(* PLC project tipper, Dassault Systèmes ControlBuild 2024x *)
(* stored: creationDateTime 2023-10-03T11:12:52-01:00 *)

(* This module simulates the behaviour of a tipper. It takes a rotation speed as input and can move actors and products that are in interaction. *)
FUNCTION_BLOCK equipment_library.tipper
  VAR_INPUT
    rotationSpeed : REAL := 0.0;
  END_VAR
  VAR_OUTPUT
    angleRotationRad : REAL := 0.0;
    incRotation : REAL := 0.0;
    angleRotationDeg : REAL := 0.0;
  END_VAR
  VAR
    status_act_prod : DINT := 0;
    m11 : REAL := 1.0;
    m12 : REAL := 0.0;
    m13 : REAL := 0.0;
    m14 : REAL := 0.0;
    m21 : REAL := 0.0;
    m22 : REAL := 1.0;
    m23 : REAL := 0.0;
    m24 : REAL := 0.0;
    m31 : REAL := 0.0;
    m32 : REAL := 0.0;
    m33 : REAL := 1.0;
    m34 : REAL := 0.0;
    m41 : REAL := 0.0;
    m42 : REAL := 0.0;
    m43 : REAL := 0.0;
    m44 : REAL := 1.0;
    incrementRotation : REAL := 0.0;
    initPosX : REAL := 0.0;
    initPosY : REAL := 0.0;
    initPosZ : REAL := 0.0;
    firstCycle : BOOL := false;
  END_VAR
  VAR CONSTANT
    fixedPositions : ARRAY[1..5] OF REAL := [0.0, 90.0, 180.0, 270.0, 360.0];
    deltaPos : REAL(0.0..45.0) := 15.0;
  END_VAR
  VAR
    d_locking : BOOL := false;
    v_d_locking : REAL := 0.0;
    d_position : BOOL := false;
    v_d_position : REAL := 0.0;
  END_VAR


ACTION C_source_code:
/* ----------------------------------------------------------------	*/
/* Type : Model of Operative Behaviour					*/
/* Category :  Actors and Products						*/
/* Author : Dassault Systemes						*/
/* Update date : June 2018							*/
/* ----------------------------------------------------------------	*/
/* This module simulates the behaviour of a tipper.			*/
/* It takes a rotation speed as input and can move actors and		*/
/* products that are in interaction.					*/
/* ----------------------------------------------------------------	*/

/* ----------------------------------------------------------------	*/
/* Save initials rotation center position	s				*/
/* ----------------------------------------------------------------	*/
if (! firstCycle) {
	initPosX = getCenterX(myself);
	initPosY = getCenterY(myself);
	initPosZ = getPositionZ(myself)+getSizeZ(myself);
	firstCycle=1;
}

/* ----------------------------------------------------------------	*/
/* Management of the rotation						*/
/* ----------------------------------------------------------------	*/
if (d_locking) 
	incrementRotation = 0;
else {
	/* Compute the increment of rotation according to the simulation clock	*/
	incrementRotation = rotationSpeed * (CLOCK_PERIOD/1000000.0) ;	
}

/* ----------------------------------------------------------------	*/
/* Request for updating the plate ring's position 			*/
/* ----------------------------------------------------------------	*/
if (d_position) {
	incrementRotation = v_d_position - angleRotationDeg;
	d_position = 0;
}

/* ----------------------------------------------------------------	*/
/* Request for align the tipper in fixed position 			*/
/* ----------------------------------------------------------------	*/
if (rotationSpeed == 0.0) {
	CB_Int i;
	CB_Float currentAngle;
	currentAngle=angleRotationDeg;  
	for (i=1; i<=5; i++) {
		if ((currentAngle- deltaPos < fixedPositions(i)) && (currentAngle+ deltaPos > fixedPositions(i))) {
			incrementRotation = fixedPositions(i) - currentAngle;
			break;
		 }
	}
}



/* ----------------------------------------------------------------	*/
/* Compute the rotation angle in degrees and in radians		*/
/* ----------------------------------------------------------------	*/
angleRotationDeg += incrementRotation;
angleRotationRad = angleRotationDeg * PI/180.0;



/* ----------------------------------------------------------------	*/
/* Output of the rotation angle for rotated actors/products		*/
/* ----------------------------------------------------------------	*/
incRotation = incrementRotation;
END_ACTION

ACTION C_header:
#ifndef PI
#define PI 3.1415926535898
#endif
END_ACTION
END_FUNCTION_BLOCK
